FUNCTION_BLOCK FB_HwRefInkStatDriveSpin EXTENDS FB_CanNodeBase
VAR_INPUT
	//Ausgänge
	nControl		AT %Q* : UINT; 	//Controlword
	nOpMode			AT %Q* : USINT;	//Mode of Operations
	nSpeed			AT %Q* : INT;	//Speed
	bDigiOut0		AT %Q* : BOOL;	//Digitaler Ausgang0
	bDigiOut1		AT %Q* : BOOL;	//Digitaler Ausgang1
	bIsInit 		: BOOL;
END_VAR
VAR_OUTPUT
	//Eingänge
	nStatus	 		AT %I* : UINT;	//Statusword
	nCurrentOpMode	AT %I* : USINT; //Aktueller Wert von Mode of Operation
	bHallSens		AT %I* : BOOL;	//Hall-Sensor
	bZSensor		AT %I* : BOOL;	//ZSensor
	nCurrentSpeed	AT %I* : INT;	//Aktuelle Drehzahl
	nCurrentVacuum : INT;
END_VAR
VAR
	timer : TON;
	nState	: USINT;
END_VAR

IF bNodeEnabled THEN
	SUPER^();
	//Vacuum abrufen alle 1s
	IF bIsInit THEN
		CASE nState OF
			0:	//Analogwert per SDO auslesen
				fbSdoRead(sADSNetID:= stAdsAdress.sNetId,nPortNr:= stAdsAdress.nPort,
						nIndex:= 16#270E, nSubIndex:= 1, nDataLength:= 4, bExecute:= TRUE);
						
				IF NOT fbSdoRead.bBusy THEN
					IF NOT fbSdoRead.bError THEN
						//Vacuum-Sensor misst den Absolutdruck.
						//Messbereich 20-400kPa (absolut) bei Ausgangsspannung 0,2V - 4,8V
						//als atmosphärischer Druck wird 100kPa angenommen
						nCurrentVacuum := REAL_TO_INT((F_YFuncX(rxMin:= 0.2, rxMax:= 4.8,
												ryMin:= 20.0, ryMax:= 400.0,
												rx:= 10.0/4095.0* DINT_TO_REAL(fbSdoRead.nData))) - 100.0);
						
						fbSdoRead(bExecute:= FALSE);
						
					END_IF
					nState := 1;
				END_IF
				
			1:	//Warten
				timer(IN:= TRUE, PT:= T#1S);
				IF timer.Q THEN
					timer(IN:= FALSE);
					nState := 0;
				END_IF
		END_CASE
		
		//LED-Anzeige (nur bei manchen Bauformen)
		IF nCurrentSpeed = 0 THEN
			bDigiOut0 := FALSE;
		ELSE
			bDigiOut0 := TRUE;
		END_IF
		
	ELSE
		nCurrentVacuum := 0;
 	END_IF
	
END_IF

END_FUNCTION_BLOCK

(* stored: Version 1.1.0.1, ProductVersion 3.1.4020.12
   POU FB_HwRefInkStatDriveSpin: Id {da497482-61e8-4d46-9bd1-e43542b9be37}, SpecialFunc None *)
